// TIA Portal V17 export
// export: Created 2025-03-07T09:16:32.0834683Z, ExportSetting WithDefaults, DisplayName Totally Integrated Automation Portal, DisplayVersion V17 Update 8, DisplayName TIA Portal Openness, DisplayVersion V17 Update 8, DisplayName TIA Portal Version Control Interface, DisplayVersion V17, DisplayName SINAMICS Startdrive Advanced, DisplayVersion V17 SP2, DisplayName SINAMICS Startdrive G110M, G120, G120C, G120D, G120P, G115D, DisplayVersion V17 SP2, DisplayName SINAMICS Startdrive G130, G150, S120, S150, SINAMICS MV, S210, DisplayVersion V17 SP2, DisplayName STEP 7 Professional, DisplayVersion V17 Update 8, DisplayName SINUMERIK ONE STEP 7 Toolbox, DisplayVersion V17 Update 12, DisplayName SINUMERIK 840D sl STEP 7 Toolbox, DisplayVersion V17 Update 12, DisplayName STEP 7 Safety, DisplayVersion V17 Update 6, DisplayName WinCC Advanced, DisplayVersion V17 Update 8
DATA_BLOCK "LBP_ParamAlarmMsgs"   // DB5
TITLE = PLC-Error / Messages / PLC errores/avisos / PLC-Fehler / Meldungen
{ S7_Optimized_Access := 'FALSE'; DB_Accessible_From_OPC_UA := 'FALSE' }
AUTHOR : SINUMERIK
FAMILY : SINUMERIK_ONE
VERSION : 6.15
// Interface between user program and LBP_GenAlarmMsgs [FC10], contains the parameter assignment of the alarms for the bit arrays in the LBP_AlarmMsgs [DB2] as fault or status message. / Interfaz entre programa de usuario y LBP_GenAlarmMsgs [FC10], contiene la asignación de parámetros de las alarmas para los arrays de bits en LBP_AlarmMsgs [DB2] como avisos de fallo o de estado. / Schnittstelle zwischen Anwenderprogramm und LBP_GenAlarmMsgs [FC10], enthält die Parameterzuordnung der Alarme für die Bit-Arrays in der LBP_AlarmMsgs [DB2] als Störungs- oder Statusmeldungen.
// stored: AutoNumber false, DBAccessibleFromOPCUA false, DBAccessibleFromWebserver true, IsOnlyStoredInLoadMemory false, IsWriteProtectedInAS false
   VAR RETAIN
      Ch1_DB2_310 : Bool := TRUE;   // (Kanäle 1-10, je 18 Bit): DB2.DBB310; Fehlermeldungen / (Channels 1-10, 18 bits each): DB2.DBB310; error messages / (Canales 1-10, cada uno 18 bits): DB2.DBB310; avisos de error
      Ch1_DB2_311 : Bool := FALSE;   // Kanal 1, DB2.DBB311; Betriebsmeldungen / Channel 1, DB2.DBB311; operating messages / Canal 1, DB2.DBB311; avisos operativos
      Ch1_DB2_312 : Bool := TRUE;   // Kanal 1, DB2.DBB312; Fehlermeldungen / Channel 1, DB2.DBB312; error messages / Canal 1, DB2.DBB312; avisos de error
      Ch1_DB2_313 : Bool := TRUE;   // Fehlermeldungen / Error messages / Avisos de error
      Ch1_DB2_314 : Bool := FALSE;   // Betriebsmeldungen / Operating messages / Avisos operativos
      Ch1_DB2_315 : Bool := FALSE;   // Betriebsmeldungen / Operating messages / Avisos operativos
      Ch1_DB2_316 : Bool := TRUE;   // Fehlermeldungen / Error messages / Avisos de error
      Ch1_DB2_317 : Bool := TRUE;   // Fehlermeldungen / Error messages / Avisos de error
      Ch1_DB2_318 : Bool := FALSE;   // Betriebsmeldungen / Operating messages / Avisos operativos
      Ch1_DB2_319 : Bool := FALSE;   // Betriebsmeldungen / Operating messages / Avisos operativos
      Ch1_DB2_320 : Bool := TRUE;   // Fehlermeldungen / Error messages / Avisos de error
      Ch1_DB2_321 : Bool := FALSE;   // Betriebsmeldungen / Operating messages / Avisos operativos
      Ch1_DB2_322 : Bool := TRUE;   // Fehlermeldungen / Error messages / Avisos de error
      Ch1_DB2_323 : Bool := FALSE;   // Betriebsmeldungen / Operating messages / Avisos operativos
      Ch1_DB2_324 : Bool := TRUE;   // Fehlermeldungen / Error messages / Avisos de error
      Ch1_DB2_325 : Bool := FALSE;   // Betriebsmeldungen / Operating messages / Avisos operativos
      Ch1_DB2_326 : Bool := TRUE;   // Fehlermeldungen / Error messages / Avisos de error
      Ch1_DB2_327 : Bool := FALSE;   // Betriebsmeldungen / Operating messages / Avisos operativos
      Ch2_DB2_328 : Bool := TRUE;   // Kanal 2, DB2.DBB328; Fehlermeldungen / Channel 2, DB2.DBB328; error messages / Canal 2, DB2.DBB328; avisos de error
      Ch2_DB2_329 : Bool := FALSE;   // Kanal 2, DB2.DBB329; Betriebsmeldungen / Channel 2, DB2.DBB329; operating messages / Canal 2, DB2.DBB329; avisos operativos
      Ch2_DB2_330 : Bool := TRUE;   // Fehlermeldungen / Error messages / Avisos de error
      Ch2_DB2_331 : Bool := TRUE;   // Fehlermeldungen / Error messages / Avisos de error
      Ch2_DB2_332 : Bool := FALSE;   // Betriebsmeldungen / Operating messages / Avisos operativos
      Ch2_DB2_333 : Bool := FALSE;   // Betriebsmeldungen / Operating messages / Avisos operativos
      Ch2_DB2_334 : Bool := TRUE;   // Fehlermeldungen / Error messages / Avisos de error
      Ch2_DB2_335 : Bool := TRUE;   // Fehlermeldungen / Error messages / Avisos de error
      Ch2_DB2_336 : Bool := FALSE;   // Betriebsmeldungen / Operating messages / Avisos operativos
      Ch2_DB2_337 : Bool := FALSE;   // Betriebsmeldungen / Operating messages / Avisos operativos
      Ch2_DB2_338 : Bool := TRUE;   // Fehlermeldungen / Error messages / Avisos de error
      Ch2_DB2_339 : Bool := FALSE;   // Betriebsmeldungen / Operating messages / Avisos operativos
      Ch2_DB2_340 : Bool := TRUE;   // Fehlermeldungen / Error messages / Avisos de error
      Ch2_DB2_341 : Bool := FALSE;   // Betriebsmeldungen / Operating messages / Avisos operativos
      Ch2_DB2_342 : Bool := TRUE;   // Fehlermeldungen / Error messages / Avisos de error
      Ch2_DB2_343 : Bool := FALSE;   // Betriebsmeldungen / Operating messages / Avisos operativos
      Ch2_DB2_344 : Bool := TRUE;   // Fehlermeldungen / Error messages / Avisos de error
      Ch2_DB2_345 : Bool := FALSE;   // Betriebsmeldungen / Operating messages / Avisos operativos
      Ch3_DB2_346 : Bool := TRUE;   // Kanal 3, DB2.DBB346; Fehlermeldungen / Channel 3, DB2.DBB346; error messages / Canal 3, DB2.DBB346; avisos de error
      Ch3_DB2_347 : Bool := FALSE;   // Kanal 3, DB2.DBB347; Betriebsmeldungen / Channel 3, DB2.DBB347; operating messages / Canal 3, DB2.DBB347; avisos operativos
      Ch3_DB2_348 : Bool := TRUE;   // Fehlermeldungen / Error messages / Avisos de error
      Ch3_DB2_349 : Bool := TRUE;   // Fehlermeldungen / Error messages / Avisos de error
      Ch3_DB2_350 : Bool := FALSE;   // Betriebsmeldungen / Operating messages / Avisos operativos
      Ch3_DB2_351 : Bool := FALSE;   // Betriebsmeldungen / Operating messages / Avisos operativos
      Ch3_DB2_352 : Bool := TRUE;   // Fehlermeldungen / Error messages / Avisos de error
      Ch3_DB2_353 : Bool := TRUE;   // Fehlermeldungen / Error messages / Avisos de error
      Ch3_DB2_354 : Bool := FALSE;   // Betriebsmeldungen / Operating messages / Avisos operativos
      Ch3_DB2_355 : Bool := FALSE;   // Betriebsmeldungen / Operating messages / Avisos operativos
      Ch3_DB2_356 : Bool := TRUE;   // Fehlermeldungen / Error messages / Avisos de error
      Ch3_DB2_357 : Bool := FALSE;   // Betriebsmeldungen / Operating messages / Avisos operativos
      Ch3_DB2_358 : Bool := TRUE;   // Fehlermeldungen / Error messages / Avisos de error
      Ch3_DB2_359 : Bool := FALSE;   // Betriebsmeldungen / Operating messages / Avisos operativos
      Ch3_DB2_360 : Bool := TRUE;   // Fehlermeldungen / Error messages / Avisos de error
      Ch3_DB2_361 : Bool := FALSE;   // Betriebsmeldungen / Operating messages / Avisos operativos
      Ch3_DB2_362 : Bool := TRUE;   // Fehlermeldungen / Error messages / Avisos de error
      Ch3_DB2_363 : Bool := FALSE;   // Betriebsmeldungen / Operating messages / Avisos operativos
      Ch4_DB2_364 : Bool := TRUE;   // Kanal 4, DB2.DBB364; Fehlermeldungen / Channel 4, DB2.DBB364; error messages / Canal 4, DB2.DBB364; avisos de error
      Ch4_DB2_365 : Bool := FALSE;   // Kanal 4, DB2.DBB365; Betriebsmeldungen / Channel 4, DB2.DBB365; operating messages / Canal 4, DB2.DBB365; avisos operativos
      Ch4_DB2_366 : Bool := TRUE;   // Fehlermeldungen / Error messages / Avisos de error
      Ch4_DB2_367 : Bool := TRUE;   // Fehlermeldungen / Error messages / Avisos de error
      Ch4_DB2_368 : Bool := FALSE;   // Betriebsmeldungen / Operating messages / Avisos operativos
      Ch4_DB2_369 : Bool := FALSE;   // Betriebsmeldungen / Operating messages / Avisos operativos
      Ch4_DB2_370 : Bool := TRUE;   // Fehlermeldungen / Error messages / Avisos de error
      Ch4_DB2_371 : Bool := TRUE;   // Fehlermeldungen / Error messages / Avisos de error
      Ch4_DB2_372 : Bool := FALSE;   // Betriebsmeldungen / Operating messages / Avisos operativos
      Ch4_DB2_373 : Bool := FALSE;   // Betriebsmeldungen / Operating messages / Avisos operativos
      Ch4_DB2_374 : Bool := TRUE;   // Fehlermeldungen / Error messages / Avisos de error
      Ch4_DB2_375 : Bool := FALSE;   // Betriebsmeldungen / Operating messages / Avisos operativos
      Ch4_DB2_376 : Bool := TRUE;   // Fehlermeldungen / Error messages / Avisos de error
      Ch4_DB2_377 : Bool := FALSE;   // Betriebsmeldungen / Operating messages / Avisos operativos
      Ch4_DB2_378 : Bool := TRUE;   // Fehlermeldungen / Error messages / Avisos de error
      Ch4_DB2_379 : Bool := FALSE;   // Betriebsmeldungen / Operating messages / Avisos operativos
      Ch4_DB2_380 : Bool := TRUE;   // Fehlermeldungen / Error messages / Avisos de error
      Ch4_DB2_381 : Bool := FALSE;   // Betriebsmeldungen / Operating messages / Avisos operativos
      Ch5_DB2_382 : Bool := TRUE;   // Kanal 5, DB2.DBB382; Fehlermeldungen / Channel 5, DB2.DBB382; error messages / Canal 5, DB2.DBB382; avisos de error
      Ch5_DB2_383 : Bool := FALSE;   // Kanal 5, DB2.DBB383; Betriebsmeldungen / Channel 5, DB2.DBB383; operating messages / Canal 5, DB2.DBB383; avisos operativos
      Ch5_DB2_384 : Bool := TRUE;   // Fehlermeldungen / Error messages / Avisos de error
      Ch5_DB2_385 : Bool := TRUE;   // Fehlermeldungen / Error messages / Avisos de error
      Ch5_DB2_386 : Bool := FALSE;   // Betriebsmeldungen / Operating messages / Avisos operativos
      Ch5_DB2_387 : Bool := FALSE;   // Betriebsmeldungen / Operating messages / Avisos operativos
      Ch5_DB2_388 : Bool := TRUE;   // Fehlermeldungen / Error messages / Avisos de error
      Ch5_DB2_389 : Bool := TRUE;   // Fehlermeldungen / Error messages / Avisos de error
      Ch5_DB2_390 : Bool := FALSE;   // Betriebsmeldungen / Operating messages / Avisos operativos
      Ch5_DB2_391 : Bool := FALSE;   // Betriebsmeldungen / Operating messages / Avisos operativos
      Ch5_DB2_392 : Bool := TRUE;   // Fehlermeldungen / Error messages / Avisos de error
      Ch5_DB2_393 : Bool := FALSE;   // Betriebsmeldungen / Operating messages / Avisos operativos
      Ch5_DB2_394 : Bool := TRUE;   // Fehlermeldungen / Error messages / Avisos de error
      Ch5_DB2_395 : Bool := FALSE;   // Betriebsmeldungen / Operating messages / Avisos operativos
      Ch5_DB2_396 : Bool := TRUE;   // Fehlermeldungen / Error messages / Avisos de error
      Ch5_DB2_397 : Bool := FALSE;   // Betriebsmeldungen / Operating messages / Avisos operativos
      Ch5_DB2_398 : Bool := TRUE;   // Fehlermeldungen / Error messages / Avisos de error
      Ch5_DB2_399 : Bool := FALSE;   // Betriebsmeldungen / Operating messages / Avisos operativos
      Ch6_DB2_400 : Bool := TRUE;   // Kanal 6, DB2.DBB400; Fehlermeldungen / Channel 6, DB2.DBB400; error messages / Canal 6, DB2.DBB400; avisos de error
      Ch6_DB2_401 : Bool := FALSE;   // Kanal 6, DB2.DBB401; Betriebsmeldungen / Channel 6, DB2.DBB401; operating messages / Canal 6, DB2.DBB401; avisos operativos
      Ch6_DB2_402 : Bool := TRUE;   // Fehlermeldungen / Error messages / Avisos de error
      Ch6_DB2_403 : Bool := TRUE;   // Fehlermeldungen / Error messages / Avisos de error
      Ch6_DB2_404 : Bool := FALSE;   // Betriebsmeldungen / Operating messages / Avisos operativos
      Ch6_DB2_405 : Bool := FALSE;   // Betriebsmeldungen / Operating messages / Avisos operativos
      Ch6_DB2_406 : Bool := TRUE;   // Fehlermeldungen / Error messages / Avisos de error
      Ch6_DB2_407 : Bool := TRUE;   // Fehlermeldungen / Error messages / Avisos de error
      Ch6_DB2_408 : Bool := FALSE;   // Betriebsmeldungen / Operating messages / Avisos operativos
      Ch6_DB2_409 : Bool := FALSE;   // Betriebsmeldungen / Operating messages / Avisos operativos
      Ch6_DB2_410 : Bool := TRUE;   // Fehlermeldungen / Error messages / Avisos de error
      Ch6_DB2_411 : Bool := FALSE;   // Betriebsmeldungen / Operating messages / Avisos operativos
      Ch6_DB2_412 : Bool := TRUE;   // Fehlermeldungen / Error messages / Avisos de error
      Ch6_DB2_413 : Bool := FALSE;   // Betriebsmeldungen / Operating messages / Avisos operativos
      Ch6_DB2_414 : Bool := TRUE;   // Fehlermeldungen / Error messages / Avisos de error
      Ch6_DB2_415 : Bool := FALSE;   // Betriebsmeldungen / Operating messages / Avisos operativos
      Ch6_DB2_416 : Bool := TRUE;   // Fehlermeldungen / Error messages / Avisos de error
      Ch6_DB2_417 : Bool := FALSE;   // Betriebsmeldungen / Operating messages / Avisos operativos
      Ch7_DB2_418 : Bool := TRUE;   // Kanal 7, DB2.DBB418; Fehlermeldungen / Channel 7, DB2.DBB418; error messages / Canal 7, DB2.DBB418; avisos de error
      Ch7_DB2_419 : Bool := FALSE;   // Kanal 7, DB2.DBB419; Betriebsmeldungen / Channel 7, DB2.DBB419; operating messages / Canal 7, DB2.DBB419; avisos operativos
      Ch7_DB2_420 : Bool := TRUE;   // Fehlermeldungen / Error messages / Avisos de error
      Ch7_DB2_421 : Bool := TRUE;   // Fehlermeldungen / Error messages / Avisos de error
      Ch7_DB2_422 : Bool := FALSE;   // Betriebsmeldungen / Operating messages / Avisos operativos
      Ch7_DB2_423 : Bool := FALSE;   // Betriebsmeldungen / Operating messages / Avisos operativos
      Ch7_DB2_424 : Bool := TRUE;   // Fehlermeldungen / Error messages / Avisos de error
      Ch7_DB2_425 : Bool := TRUE;   // Fehlermeldungen / Error messages / Avisos de error
      Ch7_DB2_426 : Bool := FALSE;   // Betriebsmeldungen / Operating messages / Avisos operativos
      Ch7_DB2_427 : Bool := FALSE;   // Betriebsmeldungen / Operating messages / Avisos operativos
      Ch7_DB2_428 : Bool := TRUE;   // Fehlermeldungen / Error messages / Avisos de error
      Ch7_DB2_429 : Bool := FALSE;   // Betriebsmeldungen / Operating messages / Avisos operativos
      Ch7_DB2_430 : Bool := TRUE;   // Fehlermeldungen / Error messages / Avisos de error
      Ch7_DB2_431 : Bool := FALSE;   // Betriebsmeldungen / Operating messages / Avisos operativos
      Ch7_DB2_432 : Bool := TRUE;   // Fehlermeldungen / Error messages / Avisos de error
      Ch7_DB2_433 : Bool := FALSE;   // Betriebsmeldungen / Operating messages / Avisos operativos
      Ch7_DB2_434 : Bool := TRUE;   // Fehlermeldungen / Error messages / Avisos de error
      Ch7_DB2_435 : Bool := FALSE;   // Betriebsmeldungen / Operating messages / Avisos operativos
      Ch8_DB2_436 : Bool := TRUE;   // Kanal 8, DB2.DBB436; Fehlermeldungen / Channel 8, DB2.DBB436; error messages / Canal 8, DB2.DBB436; avisos de error
      Ch8_DB2_437 : Bool := FALSE;   // Kanal 8, DB2.DBB437; Betriebsmeldungen / Channel 8, DB2.DBB437; operating messages / Canal 8, DB2.DBB437; avisos operativos
      Ch8_DB2_438 : Bool := TRUE;   // Fehlermeldungen / Error messages / Avisos de error
      Ch8_DB2_439 : Bool := TRUE;   // Fehlermeldungen / Error messages / Avisos de error
      Ch8_DB2_440 : Bool := FALSE;   // Betriebsmeldungen / Operating messages / Avisos operativos
      Ch8_DB2_441 : Bool := FALSE;   // Betriebsmeldungen / Operating messages / Avisos operativos
      Ch8_DB2_442 : Bool := TRUE;   // Fehlermeldungen / Error messages / Avisos de error
      Ch8_DB2_443 : Bool := TRUE;   // Fehlermeldungen / Error messages / Avisos de error
      Ch8_DB2_444 : Bool := FALSE;   // Betriebsmeldungen / Operating messages / Avisos operativos
      Ch8_DB2_445 : Bool := FALSE;   // Betriebsmeldungen / Operating messages / Avisos operativos
      Ch8_DB2_446 : Bool := TRUE;   // Fehlermeldungen / Error messages / Avisos de error
      Ch8_DB2_447 : Bool := FALSE;   // Betriebsmeldungen / Operating messages / Avisos operativos
      Ch8_DB2_448 : Bool := TRUE;   // Fehlermeldungen / Error messages / Avisos de error
      Ch8_DB2_449 : Bool := FALSE;   // Betriebsmeldungen / Operating messages / Avisos operativos
      Ch8_DB2_450 : Bool := TRUE;   // Fehlermeldungen / Error messages / Avisos de error
      Ch8_DB2_451 : Bool := FALSE;   // Betriebsmeldungen / Operating messages / Avisos operativos
      Ch8_DB2_452 : Bool := TRUE;   // Fehlermeldungen / Error messages / Avisos de error
      Ch8_DB2_453 : Bool := FALSE;   // Betriebsmeldungen / Operating messages / Avisos operativos
      Ch9_DB2_454 : Bool := TRUE;   // Kanal 9, DB2.DBB454; Fehlermeldungen / Channel 9, DB2.DBB454; error messages / Canal 9, DB2.DBB454; avisos de error
      Ch9_DB2_455 : Bool := FALSE;   // Kanal 9, DB2.DBB455; Betriebsmeldungen / Channel 9, DB2.DBB455; operating messages / Canal 9, DB2.DBB455; avisos operativos
      Ch9_DB2_456 : Bool := TRUE;   // Fehlermeldungen / Error messages / Avisos de error
      Ch9_DB2_457 : Bool := TRUE;   // Fehlermeldungen / Error messages / Avisos de error
      Ch9_DB2_458 : Bool := FALSE;   // Betriebsmeldungen / Operating messages / Avisos operativos
      Ch9_DB2_459 : Bool := FALSE;   // Betriebsmeldungen / Operating messages / Avisos operativos
      Ch9_DB2_460 : Bool := TRUE;   // Fehlermeldungen / Error messages / Avisos de error
      Ch9_DB2_461 : Bool := TRUE;   // Fehlermeldungen / Error messages / Avisos de error
      Ch9_DB2_462 : Bool := FALSE;   // Betriebsmeldungen / Operating messages / Avisos operativos
      Ch9_DB2_463 : Bool := FALSE;   // Betriebsmeldungen / Operating messages / Avisos operativos
      Ch9_DB2_464 : Bool := TRUE;   // Fehlermeldungen / Error messages / Avisos de error
      Ch9_DB2_465 : Bool := FALSE;   // Betriebsmeldungen / Operating messages / Avisos operativos
      Ch9_DB2_466 : Bool := TRUE;   // Fehlermeldungen / Error messages / Avisos de error
      Ch9_DB2_467 : Bool := FALSE;   // Betriebsmeldungen / Operating messages / Avisos operativos
      Ch9_DB2_468 : Bool := TRUE;   // Fehlermeldungen / Error messages / Avisos de error
      Ch9_DB2_469 : Bool := FALSE;   // Betriebsmeldungen / Operating messages / Avisos operativos
      Ch9_DB2_470 : Bool := TRUE;   // Fehlermeldungen / Error messages / Avisos de error
      Ch9_DB2_471 : Bool := FALSE;   // Betriebsmeldungen / Operating messages / Avisos operativos
      Ch10_DB2_472 : Bool := TRUE;   // Kanal 10, DB2.DBB472; Fehlermeldungen / Channel 10, DB2.DBB472; error messages / Canal 10, DB2.DBB472; avisos de error
      Ch10_DB2_473 : Bool := FALSE;   // Kanal 10, DB2.DBB473; Betriebsmeldungen / Channel 10, DB2.DBB473; operating messages / Canal 10, DB2.DBB473; avisos operativos
      Ch10_DB2_474 : Bool := TRUE;   // Fehlermeldungen / Error messages / Avisos de error
      Ch10_DB2_475 : Bool := TRUE;   // Fehlermeldungen / Error messages / Avisos de error
      Ch10_DB2_476 : Bool := FALSE;   // Betriebsmeldungen / Operating messages / Avisos operativos
      Ch10_DB2_477 : Bool := FALSE;   // Betriebsmeldungen / Operating messages / Avisos operativos
      Ch10_DB2_478 : Bool := TRUE;   // Fehlermeldungen / Error messages / Avisos de error
      Ch10_DB2_479 : Bool := TRUE;   // Fehlermeldungen / Error messages / Avisos de error
      Ch10_DB2_480 : Bool := FALSE;   // Betriebsmeldungen / Operating messages / Avisos operativos
      Ch10_DB2_481 : Bool := FALSE;   // Betriebsmeldungen / Operating messages / Avisos operativos
      Ch10_DB2_482 : Bool := TRUE;   // Fehlermeldungen / Error messages / Avisos de error
      Ch10_DB2_483 : Bool := FALSE;   // Betriebsmeldungen / Operating messages / Avisos operativos
      Ch10_DB2_484 : Bool := TRUE;   // Fehlermeldungen / Error messages / Avisos de error
      Ch10_DB2_485 : Bool := FALSE;   // Betriebsmeldungen / Operating messages / Avisos operativos
      Ch10_DB2_486 : Bool := TRUE;   // Fehlermeldungen / Error messages / Avisos de error
      Ch10_DB2_487 : Bool := FALSE;   // Betriebsmeldungen / Operating messages / Avisos operativos
      Ch10_DB2_488 : Bool := TRUE;   // Fehlermeldungen / Error messages / Avisos de error
      Ch10_DB2_489 : Bool := FALSE;   // Betriebsmeldungen / Operating messages / Avisos operativos
      Ax1_DB2_490 : Bool := TRUE;   // (Achsen/Spindeln 1-31, je 2 Bit): DB2.DBB490; Fehlermeldungen / (Axes/Spindles 1-31, 2 bits each): DB2.DBB490; error messages / (Ejes/cabezales 1-31, cada uno 2 bits): DB2.DBB490; avisos de error
      Ax1_DB2_491 : Bool := FALSE;   // Achse/Spindel 1, DB2.DBB491; Betriebsmeldungen / Axis/Spindle 1, DB2.DBB491; operating messages / Eje/cabezal 1, DB2.DBB491; avisos operativos
      Ax2_DB2_492 : Bool := TRUE;   // Achse/Spindel 2, DB2.DBB492; Fehlermeldungen / Axis/Spindle 2, DB2.DBB492; error messages / Eje/cabezal 2, DB2.DBB492; avisos de error
      Ax2_DB2_493 : Bool := FALSE;   // Achse/Spindel 2, DB2.DBB493; Betriebsmeldungen / Axis/Spindle 2, DB2.DBB493; operating messages / Eje/cabezal 2, DB2.DBB493; avisos operativos
      Ax3_DB2_494 : Bool := TRUE;   // Fehlermeldungen / Error messages / Avisos de error
      Ax3_DB2_495 : Bool := FALSE;   // Betriebsmeldungen / Operating messages / Avisos operativos
      Ax4_DB2_496 : Bool := TRUE;   // Fehlermeldungen / Error messages / Avisos de error
      Ax4_DB2_497 : Bool := FALSE;   // Betriebsmeldungen / Operating messages / Avisos operativos
      Ax5_DB2_498 : Bool := TRUE;   // Fehlermeldungen / Error messages / Avisos de error
      Ax5_DB2_499 : Bool := FALSE;   // Betriebsmeldungen / Operating messages / Avisos operativos
      Ax6_DB2_500 : Bool := TRUE;   // Fehlermeldungen / Error messages / Avisos de error
      Ax6_DB2_501 : Bool := FALSE;   // Betriebsmeldungen / Operating messages / Avisos operativos
      Ax7_DB2_502 : Bool := TRUE;   // Fehlermeldungen / Error messages / Avisos de error
      Ax7_DB2_503 : Bool := FALSE;   // Betriebsmeldungen / Operating messages / Avisos operativos
      Ax8_DB2_504 : Bool := TRUE;   // Fehlermeldungen / Error messages / Avisos de error
      Ax8_DB2_505 : Bool := FALSE;   // Betriebsmeldungen / Operating messages / Avisos operativos
      Ax9_DB2_506 : Bool := TRUE;   // Fehlermeldungen / Error messages / Avisos de error
      Ax9_DB2_507 : Bool := FALSE;   // Betriebsmeldungen / Operating messages / Avisos operativos
      Ax10_DB2_508 : Bool := TRUE;   // Fehlermeldungen / Error messages / Avisos de error
      Ax10_DB2_509 : Bool := FALSE;   // Betriebsmeldungen / Operating messages / Avisos operativos
      Ax11_DB2_510 : Bool := TRUE;   // Fehlermeldungen / Error messages / Avisos de error
      Ax11_DB2_511 : Bool := FALSE;   // Betriebsmeldungen / Operating messages / Avisos operativos
      Ax12_DB2_512 : Bool := TRUE;   // Fehlermeldungen / Error messages / Avisos de error
      Ax12_DB2_513 : Bool := FALSE;   // Betriebsmeldungen / Operating messages / Avisos operativos
      Ax13_DB2_514 : Bool := TRUE;   // Fehlermeldungen / Error messages / Avisos de error
      Ax13_DB2_515 : Bool := FALSE;   // Betriebsmeldungen / Operating messages / Avisos operativos
      Ax14_DB2_516 : Bool := TRUE;   // Fehlermeldungen / Error messages / Avisos de error
      Ax14_DB2_517 : Bool := FALSE;   // Betriebsmeldungen / Operating messages / Avisos operativos
      Ax15_DB2_518 : Bool := TRUE;   // Fehlermeldungen / Error messages / Avisos de error
      Ax15_DB2_519 : Bool := FALSE;   // Betriebsmeldungen / Operating messages / Avisos operativos
      Ax16_DB2_520 : Bool := TRUE;   // Fehlermeldungen / Error messages / Avisos de error
      Ax16_DB2_521 : Bool := FALSE;   // Betriebsmeldungen / Operating messages / Avisos operativos
      Ax17_DB2_522 : Bool := TRUE;   // Fehlermeldungen / Error messages / Avisos de error
      Ax17_DB2_523 : Bool := FALSE;   // Betriebsmeldungen / Operating messages / Avisos operativos
      Ax18_DB2_524 : Bool := TRUE;   // Fehlermeldungen / Error messages / Avisos de error
      Ax18_DB2_525 : Bool := FALSE;   // Betriebsmeldungen / Operating messages / Avisos operativos
      Ax19_DB2_526 : Bool := TRUE;   // Fehlermeldungen / Error messages / Avisos de error
      Ax19_DB2_527 : Bool := FALSE;   // Betriebsmeldungen / Operating messages / Avisos operativos
      Ax20_DB2_528 : Bool := TRUE;   // Fehlermeldungen / Error messages / Avisos de error
      Ax20_DB2_529 : Bool := FALSE;   // Betriebsmeldungen / Operating messages / Avisos operativos
      Ax21_DB2_530 : Bool := TRUE;   // Fehlermeldungen / Error messages / Avisos de error
      Ax21_DB2_531 : Bool := FALSE;   // Betriebsmeldungen / Operating messages / Avisos operativos
      Ax22_DB2_532 : Bool := TRUE;   // Fehlermeldungen / Error messages / Avisos de error
      Ax22_DB2_533 : Bool := FALSE;   // Betriebsmeldungen / Operating messages / Avisos operativos
      Ax23_DB2_534 : Bool := TRUE;   // Fehlermeldungen / Error messages / Avisos de error
      Ax23_DB2_535 : Bool := FALSE;   // Betriebsmeldungen / Operating messages / Avisos operativos
      Ax24_DB2_536 : Bool := TRUE;   // Fehlermeldungen / Error messages / Avisos de error
      Ax24_DB2_537 : Bool := FALSE;   // Betriebsmeldungen / Operating messages / Avisos operativos
      Ax25_DB2_538 : Bool := TRUE;   // Fehlermeldungen / Error messages / Avisos de error
      Ax25_DB2_539 : Bool := FALSE;   // Betriebsmeldungen / Operating messages / Avisos operativos
      Ax26_DB2_540 : Bool := TRUE;   // Fehlermeldungen / Error messages / Avisos de error
      Ax26_DB2_541 : Bool := FALSE;   // Betriebsmeldungen / Operating messages / Avisos operativos
      Ax27_DB2_542 : Bool := TRUE;   // Fehlermeldungen / Error messages / Avisos de error
      Ax27_DB2_543 : Bool := FALSE;   // Betriebsmeldungen / Operating messages / Avisos operativos
      Ax28_DB2_544 : Bool := TRUE;   // Fehlermeldungen / Error messages / Avisos de error
      Ax28_DB2_545 : Bool := FALSE;   // Betriebsmeldungen / Operating messages / Avisos operativos
      Ax29_DB2_546 : Bool := TRUE;   // Fehlermeldungen / Error messages / Avisos de error
      Ax29_DB2_547 : Bool := FALSE;   // Betriebsmeldungen / Operating messages / Avisos operativos
      Ax30_DB2_548 : Bool := TRUE;   // Fehlermeldungen / Error messages / Avisos de error
      Ax30_DB2_549 : Bool := FALSE;   // Betriebsmeldungen / Operating messages / Avisos operativos
      Ax31_DB2_550 : Bool := TRUE;   // Fehlermeldungen / Error messages / Avisos de error
      Ax31_DB2_551 : Bool := FALSE;   // Betriebsmeldungen / Operating messages / Avisos operativos
      Bit30_2 : Bool := FALSE;   // Reserviert / Reserved / Reservado
      Bit30_3 : Bool := FALSE;   // Reserviert / Reserved / Reservado
      User0_DB2_554 : Bool := TRUE;   // (Anwender-Datenbereiche 0-31, je 8 Bit): DB2.DBB554; Fehlermeldungen / (User data areas 0-31, 8 bits each): DB2.DBB554; error messages / (Áreas de datos de usuario 0-31, cada una 8 bits): DB2.DBB554; avisos de error
      User0_DB2_555 : Bool := TRUE;   // UserDataArea 0, DB2.DBB555; Fehlermeldungen / UserDataArea 0, DB2.DBB555; error messages / UserDataArea 0, DB2.DBB555; avisos de error
      User0_DB2_556 : Bool := TRUE;   // Fehlermeldungen / Error messages / Avisos de error
      User0_DB2_557 : Bool := TRUE;   // Fehlermeldungen / Error messages / Avisos de error
      User0_DB2_558 : Bool := FALSE;   // Betriebsmeldungen / Operating messages / Avisos operativos
      User0_DB2_559 : Bool := FALSE;   // Betriebsmeldungen / Operating messages / Avisos operativos
      User0_DB2_560 : Bool := FALSE;   // Betriebsmeldungen / Operating messages / Avisos operativos
      User0_DB2_561 : Bool := FALSE;   // Betriebsmeldungen / Operating messages / Avisos operativos
      User1_DB2_562 : Bool := TRUE;   // UserDataArea 1, DB2.DBB562; Fehlermeldungen / UserDataArea 1, DB2.DBB562; error messages / UserDataArea 1, DB2.DBB562; avisos de error
      User1_DB2_563 : Bool := TRUE;   // Fehlermeldungen / Error messages / Avisos de error
      User1_DB2_564 : Bool := TRUE;   // Fehlermeldungen / Error messages / Avisos de error
      User1_DB2_565 : Bool := TRUE;   // Fehlermeldungen / Error messages / Avisos de error
      User1_DB2_566 : Bool := FALSE;   // Betriebsmeldungen / Operating messages / Avisos operativos
      User1_DB2_567 : Bool := FALSE;   // Betriebsmeldungen / Operating messages / Avisos operativos
      User1_DB2_568 : Bool := FALSE;   // Betriebsmeldungen / Operating messages / Avisos operativos
      User1_DB2_569 : Bool := FALSE;   // Betriebsmeldungen / Operating messages / Avisos operativos
      User2_DB2_570 : Bool := TRUE;   // UserDataArea 2, DB2.DBB570; Fehlermeldungen / UserDataArea 2, DB2.DBB570; error messages / UserDataArea 2, DB2.DBB570; avisos de error
      User2_DB2_571 : Bool := TRUE;   // Fehlermeldungen / Error messages / Avisos de error
      User2_DB2_572 : Bool := TRUE;   // Fehlermeldungen / Error messages / Avisos de error
      User2_DB2_573 : Bool := TRUE;   // Fehlermeldungen / Error messages / Avisos de error
      User2_DB2_574 : Bool := FALSE;   // Betriebsmeldungen / Operating messages / Avisos operativos
      User2_DB2_575 : Bool := FALSE;   // Betriebsmeldungen / Operating messages / Avisos operativos
      User2_DB2_576 : Bool := FALSE;   // Betriebsmeldungen / Operating messages / Avisos operativos
      User2_DB2_577 : Bool := FALSE;   // Betriebsmeldungen / Operating messages / Avisos operativos
      User3_DB2_578 : Bool := TRUE;   // UserDataArea 3, DB2.DBB578; Fehlermeldungen / UserDataArea 3, DB2.DBB578; error messages / UserDataArea 3, DB2.DBB578; avisos de error
      User3_DB2_579 : Bool := TRUE;   // Fehlermeldungen / Error messages / Avisos de error
      User3_DB2_580 : Bool := TRUE;   // Fehlermeldungen / Error messages / Avisos de error
      User3_DB2_581 : Bool := TRUE;   // Fehlermeldungen / Error messages / Avisos de error
      User3_DB2_582 : Bool := FALSE;   // Betriebsmeldungen / Operating messages / Avisos operativos
      User3_DB2_583 : Bool := FALSE;   // Betriebsmeldungen / Operating messages / Avisos operativos
      User3_DB2_584 : Bool := FALSE;   // Betriebsmeldungen / Operating messages / Avisos operativos
      User3_DB2_585 : Bool := FALSE;   // Betriebsmeldungen / Operating messages / Avisos operativos
      User4_DB2_586 : Bool := TRUE;   // UserDataArea 4, DB2.DBB586; Fehlermeldungen / UserDataArea 4, DB2.DBB586; error messages / UserDataArea 4, DB2.DBB586; avisos de error
      User4_DB2_587 : Bool := TRUE;   // Fehlermeldungen / Error messages / Avisos de error
      User4_DB2_588 : Bool := TRUE;   // Fehlermeldungen / Error messages / Avisos de error
      User4_DB2_589 : Bool := TRUE;   // Fehlermeldungen / Error messages / Avisos de error
      User4_DB2_590 : Bool := FALSE;   // Betriebsmeldungen / Operating messages / Avisos operativos
      User4_DB2_591 : Bool := FALSE;   // Betriebsmeldungen / Operating messages / Avisos operativos
      User4_DB2_592 : Bool := FALSE;   // Betriebsmeldungen / Operating messages / Avisos operativos
      User4_DB2_593 : Bool := FALSE;   // Betriebsmeldungen / Operating messages / Avisos operativos
      User5_DB2_594 : Bool := TRUE;   // UserDataArea 5, DB2.DBB594; Fehlermeldungen / UserDataArea 5, DB2.DBB594; error messages / UserDataArea 5, DB2.DBB594; avisos de error
      User5_DB2_595 : Bool := TRUE;   // Fehlermeldungen / Error messages / Avisos de error
      User5_DB2_596 : Bool := TRUE;   // Fehlermeldungen / Error messages / Avisos de error
      User5_DB2_597 : Bool := TRUE;   // Fehlermeldungen / Error messages / Avisos de error
      User5_DB2_598 : Bool := FALSE;   // Betriebsmeldungen / Operating messages / Avisos operativos
      User5_DB2_599 : Bool := FALSE;   // Betriebsmeldungen / Operating messages / Avisos operativos
      User5_DB2_600 : Bool := FALSE;   // Betriebsmeldungen / Operating messages / Avisos operativos
      User5_DB2_601 : Bool := FALSE;   // Betriebsmeldungen / Operating messages / Avisos operativos
      User6_DB2_602 : Bool := TRUE;   // UserDataArea 6, DB2.DBB602; Fehlermeldungen / UserDataArea 6, DB2.DBB602; error messages / UserDataArea 6, DB2.DBB602; avisos de error
      User6_DB2_603 : Bool := TRUE;   // Fehlermeldungen / Error messages / Avisos de error
      User6_DB2_604 : Bool := TRUE;   // Fehlermeldungen / Error messages / Avisos de error
      User6_DB2_605 : Bool := TRUE;   // Fehlermeldungen / Error messages / Avisos de error
      User6_DB2_606 : Bool := FALSE;   // Betriebsmeldungen / Operating messages / Avisos operativos
      User6_DB2_607 : Bool := FALSE;   // Betriebsmeldungen / Operating messages / Avisos operativos
      User6_DB2_608 : Bool := FALSE;   // Betriebsmeldungen / Operating messages / Avisos operativos
      User6_DB2_609 : Bool := FALSE;   // Betriebsmeldungen / Operating messages / Avisos operativos
      User7_DB2_610 : Bool := TRUE;   // UserDataArea 7, DB2.DBB610; Fehlermeldungen / UserDataArea 7, DB2.DBB610; error messages / UserDataArea 7, DB2.DBB610; avisos de error
      User7_DB2_611 : Bool := TRUE;   // Fehlermeldungen / Error messages / Avisos de error
      User7_DB2_612 : Bool := TRUE;   // Fehlermeldungen / Error messages / Avisos de error
      User7_DB2_613 : Bool := TRUE;   // Fehlermeldungen / Error messages / Avisos de error
      User7_DB2_614 : Bool := FALSE;   // Betriebsmeldungen / Operating messages / Avisos operativos
      User7_DB2_615 : Bool := FALSE;   // Betriebsmeldungen / Operating messages / Avisos operativos
      User7_DB2_616 : Bool := FALSE;   // Betriebsmeldungen / Operating messages / Avisos operativos
      User7_DB2_617 : Bool := FALSE;   // Betriebsmeldungen / Operating messages / Avisos operativos
      User8_DB2_618 : Bool := TRUE;   // UserDataArea 8, DB2.DBB618; Fehlermeldungen / UserDataArea 8, DB2.DBB618; error messages / UserDataArea 8, DB2.DBB618; avisos de error
      User8_DB2_619 : Bool := TRUE;   // Fehlermeldungen / Error messages / Avisos de error
      User8_DB2_620 : Bool := TRUE;   // Fehlermeldungen / Error messages / Avisos de error
      User8_DB2_621 : Bool := TRUE;   // Fehlermeldungen / Error messages / Avisos de error
      User8_DB2_622 : Bool := FALSE;   // Betriebsmeldungen / Operating messages / Avisos operativos
      User8_DB2_623 : Bool := FALSE;   // Betriebsmeldungen / Operating messages / Avisos operativos
      User8_DB2_624 : Bool := FALSE;   // Betriebsmeldungen / Operating messages / Avisos operativos
      User8_DB2_625 : Bool := FALSE;   // Betriebsmeldungen / Operating messages / Avisos operativos
      User9_DB2_626 : Bool := TRUE;   // UserDataArea 9, DB2.DBB626; Fehlermeldungen / UserDataArea 9, DB2.DBB626; error messages / UserDataArea 9, DB2.DBB626; avisos de error
      User9_DB2_627 : Bool := TRUE;   // Fehlermeldungen / Error messages / Avisos de error
      User9_DB2_628 : Bool := TRUE;   // Fehlermeldungen / Error messages / Avisos de error
      User9_DB2_629 : Bool := TRUE;   // Fehlermeldungen / Error messages / Avisos de error
      User9_DB2_630 : Bool := FALSE;   // Betriebsmeldungen / Operating messages / Avisos operativos
      User9_DB2_631 : Bool := FALSE;   // Betriebsmeldungen / Operating messages / Avisos operativos
      User9_DB2_632 : Bool := FALSE;   // Betriebsmeldungen / Operating messages / Avisos operativos
      User9_DB2_633 : Bool := FALSE;   // Betriebsmeldungen / Operating messages / Avisos operativos
      User10_DB2_634 : Bool := TRUE;   // UserDataArea 10, DB2.DBB634; Fehlermeldungen / UserDataArea 10, DB2.DBB634; error messages / UserDataArea 10, DB2.DBB634; avisos de error
      User10_DB2_635 : Bool := TRUE;   // Fehlermeldungen / Error messages / Avisos de error
      User10_DB2_636 : Bool := TRUE;   // Fehlermeldungen / Error messages / Avisos de error
      User10_DB2_637 : Bool := TRUE;   // Fehlermeldungen / Error messages / Avisos de error
      User10_DB2_638 : Bool := FALSE;   // Betriebsmeldungen / Operating messages / Avisos operativos
      User10_DB2_639 : Bool := FALSE;   // Betriebsmeldungen / Operating messages / Avisos operativos
      User10_DB2_640 : Bool := FALSE;   // Betriebsmeldungen / Operating messages / Avisos operativos
      User10_DB2_641 : Bool := FALSE;   // Betriebsmeldungen / Operating messages / Avisos operativos
      User11_DB2_642 : Bool := TRUE;   // UserDataArea 11, DB2.DBB642; Fehlermeldungen / UserDataArea 11, DB2.DBB642; error messages / UserDataArea 11, DB2.DBB642; avisos de error
      User11_DB2_643 : Bool := TRUE;   // Fehlermeldungen / Error messages / Avisos de error
      User11_DB2_644 : Bool := TRUE;   // Fehlermeldungen / Error messages / Avisos de error
      User11_DB2_645 : Bool := TRUE;   // Fehlermeldungen / Error messages / Avisos de error
      User11_DB2_646 : Bool := FALSE;   // Betriebsmeldungen / Operating messages / Avisos operativos
      User11_DB2_647 : Bool := FALSE;   // Betriebsmeldungen / Operating messages / Avisos operativos
      User11_DB2_648 : Bool := FALSE;   // Betriebsmeldungen / Operating messages / Avisos operativos
      User11_DB2_649 : Bool := FALSE;   // Betriebsmeldungen / Operating messages / Avisos operativos
      User12_DB2_650 : Bool := TRUE;   // UserDataArea 12, DB2.DBB650; Fehlermeldungen / UserDataArea 12, DB2.DBB650; error messages / UserDataArea 12, DB2.DBB650; avisos de error
      User12_DB2_651 : Bool := TRUE;   // Fehlermeldungen / Error messages / Avisos de error
      User12_DB2_652 : Bool := TRUE;   // Fehlermeldungen / Error messages / Avisos de error
      User12_DB2_653 : Bool := TRUE;   // Fehlermeldungen / Error messages / Avisos de error
      User12_DB2_654 : Bool := FALSE;   // Betriebsmeldungen / Operating messages / Avisos operativos
      User12_DB2_655 : Bool := FALSE;   // Betriebsmeldungen / Operating messages / Avisos operativos
      User12_DB2_656 : Bool := FALSE;   // Betriebsmeldungen / Operating messages / Avisos operativos
      User12_DB2_657 : Bool := FALSE;   // Betriebsmeldungen / Operating messages / Avisos operativos
      User13_DB2_658 : Bool := TRUE;   // UserDataArea 13, DB2.DBB658; Fehlermeldungen / UserDataArea 13, DB2.DBB658; error messages / UserDataArea 13, DB2.DBB658; avisos de error
      User13_DB2_659 : Bool := TRUE;   // Fehlermeldungen / Error messages / Avisos de error
      User13_DB2_660 : Bool := TRUE;   // Fehlermeldungen / Error messages / Avisos de error
      User13_DB2_661 : Bool := TRUE;   // Fehlermeldungen / Error messages / Avisos de error
      User13_DB2_662 : Bool := FALSE;   // Betriebsmeldungen / Operating messages / Avisos operativos
      User13_DB2_663 : Bool := FALSE;   // Betriebsmeldungen / Operating messages / Avisos operativos
      User13_DB2_664 : Bool := FALSE;   // Betriebsmeldungen / Operating messages / Avisos operativos
      User13_DB2_665 : Bool := FALSE;   // Betriebsmeldungen / Operating messages / Avisos operativos
      User14_DB2_666 : Bool := TRUE;   // UserDataArea 14, DB2.DBB666; Fehlermeldungen / UserDataArea 14, DB2.DBB666; error messages / UserDataArea 14, DB2.DBB666; avisos de error
      User14_DB2_667 : Bool := TRUE;   // Fehlermeldungen / Error messages / Avisos de error
      User14_DB2_668 : Bool := TRUE;   // Fehlermeldungen / Error messages / Avisos de error
      User14_DB2_669 : Bool := TRUE;   // Fehlermeldungen / Error messages / Avisos de error
      User14_DB2_670 : Bool := FALSE;   // Betriebsmeldungen / Operating messages / Avisos operativos
      User14_DB2_671 : Bool := FALSE;   // Betriebsmeldungen / Operating messages / Avisos operativos
      User14_DB2_672 : Bool := FALSE;   // Betriebsmeldungen / Operating messages / Avisos operativos
      User14_DB2_673 : Bool := FALSE;   // Betriebsmeldungen / Operating messages / Avisos operativos
      User15_DB2_674 : Bool := TRUE;   // UserDataArea 15, DB2.DBB674; Fehlermeldungen / UserDataArea 15, DB2.DBB674; error messages / UserDataArea 15, DB2.DBB674; avisos de error
      User15_DB2_675 : Bool := TRUE;   // Fehlermeldungen / Error messages / Avisos de error
      User15_DB2_676 : Bool := TRUE;   // Fehlermeldungen / Error messages / Avisos de error
      User15_DB2_677 : Bool := TRUE;   // Fehlermeldungen / Error messages / Avisos de error
      User15_DB2_678 : Bool := FALSE;   // Betriebsmeldungen / Operating messages / Avisos operativos
      User15_DB2_679 : Bool := FALSE;   // Betriebsmeldungen / Operating messages / Avisos operativos
      User15_DB2_680 : Bool := FALSE;   // Betriebsmeldungen / Operating messages / Avisos operativos
      User15_DB2_681 : Bool := FALSE;   // Betriebsmeldungen / Operating messages / Avisos operativos
      User16_DB2_682 : Bool := TRUE;   // UserDataArea 16, DB2.DBB682; Fehlermeldungen / UserDataArea 16, DB2.DBB682; error messages / UserDataArea 16, DB2.DBB682; avisos de error
      User16_DB2_683 : Bool := TRUE;   // Fehlermeldungen / Error messages / Avisos de error
      User16_DB2_684 : Bool := TRUE;   // Fehlermeldungen / Error messages / Avisos de error
      User16_DB2_685 : Bool := TRUE;   // Fehlermeldungen / Error messages / Avisos de error
      User16_DB2_686 : Bool := FALSE;   // Betriebsmeldungen / Operating messages / Avisos operativos
      User16_DB2_687 : Bool := FALSE;   // Betriebsmeldungen / Operating messages / Avisos operativos
      User16_DB2_688 : Bool := FALSE;   // Betriebsmeldungen / Operating messages / Avisos operativos
      User16_DB2_689 : Bool := FALSE;   // Betriebsmeldungen / Operating messages / Avisos operativos
      User17_DB2_690 : Bool := TRUE;   // UserDataArea 17, DB2.DBB690; Fehlermeldungen / UserDataArea 17, DB2.DBB690; error messages / UserDataArea 17, DB2.DBB690; avisos de error
      User17_DB2_691 : Bool := TRUE;   // Fehlermeldungen / Error messages / Avisos de error
      User17_DB2_692 : Bool := TRUE;   // Fehlermeldungen / Error messages / Avisos de error
      User17_DB2_693 : Bool := TRUE;   // Fehlermeldungen / Error messages / Avisos de error
      User17_DB2_694 : Bool := FALSE;   // Betriebsmeldungen / Operating messages / Avisos operativos
      User17_DB2_695 : Bool := FALSE;   // Betriebsmeldungen / Operating messages / Avisos operativos
      User17_DB2_696 : Bool := FALSE;   // Betriebsmeldungen / Operating messages / Avisos operativos
      User17_DB2_697 : Bool := FALSE;   // Betriebsmeldungen / Operating messages / Avisos operativos
      User18_DB2_698 : Bool := TRUE;   // UserDataArea 18, DB2.DBB698; Fehlermeldungen / UserDataArea 18, DB2.DBB698; error messages / UserDataArea 18, DB2.DBB698; avisos de error
      User18_DB2_699 : Bool := TRUE;   // Fehlermeldungen / Error messages / Avisos de error
      User18_DB2_700 : Bool := TRUE;   // Fehlermeldungen / Error messages / Avisos de error
      User18_DB2_701 : Bool := TRUE;   // Fehlermeldungen / Error messages / Avisos de error
      User18_DB2_702 : Bool := FALSE;   // Betriebsmeldungen / Operating messages / Avisos operativos
      User18_DB2_703 : Bool := FALSE;   // Betriebsmeldungen / Operating messages / Avisos operativos
      User18_DB2_704 : Bool := FALSE;   // Betriebsmeldungen / Operating messages / Avisos operativos
      User18_DB2_705 : Bool := FALSE;   // Betriebsmeldungen / Operating messages / Avisos operativos
      User19_DB2_706 : Bool := TRUE;   // UserDataArea 19, DB2.DBB706; Fehlermeldungen / UserDataArea 19, DB2.DBB706; error messages / UserDataArea 19, DB2.DBB706; avisos de error
      User19_DB2_707 : Bool := TRUE;   // Fehlermeldungen / Error messages / Avisos de error
      User19_DB2_708 : Bool := TRUE;   // Fehlermeldungen / Error messages / Avisos de error
      User19_DB2_709 : Bool := TRUE;   // Fehlermeldungen / Error messages / Avisos de error
      User19_DB2_710 : Bool := FALSE;   // Betriebsmeldungen / Operating messages / Avisos operativos
      User19_DB2_711 : Bool := FALSE;   // Betriebsmeldungen / Operating messages / Avisos operativos
      User19_DB2_712 : Bool := FALSE;   // Betriebsmeldungen / Operating messages / Avisos operativos
      User19_DB2_713 : Bool := FALSE;   // Betriebsmeldungen / Operating messages / Avisos operativos
      User20_DB2_714 : Bool := TRUE;   // UserDataArea 20, DB2.DBB714; Fehlermeldungen / UserDataArea 20, DB2.DBB714; error messages / UserDataArea 20, DB2.DBB714; avisos de error
      User20_DB2_715 : Bool := TRUE;   // Fehlermeldungen / Error messages / Avisos de error
      User20_DB2_716 : Bool := TRUE;   // Fehlermeldungen / Error messages / Avisos de error
      User20_DB2_717 : Bool := TRUE;   // Fehlermeldungen / Error messages / Avisos de error
      User20_DB2_718 : Bool := FALSE;   // Betriebsmeldungen / Operating messages / Avisos operativos
      User20_DB2_719 : Bool := FALSE;   // Betriebsmeldungen / Operating messages / Avisos operativos
      User20_DB2_720 : Bool := FALSE;   // Betriebsmeldungen / Operating messages / Avisos operativos
      User20_DB2_721 : Bool := FALSE;   // Betriebsmeldungen / Operating messages / Avisos operativos
      User21_DB2_722 : Bool := TRUE;   // UserDataArea 21, DB2.DBB722; Fehlermeldungen / UserDataArea 21, DB2.DBB722; error messages / UserDataArea 21, DB2.DBB722; avisos de error
      User21_DB2_723 : Bool := TRUE;   // Fehlermeldungen / Error messages / Avisos de error
      User21_DB2_724 : Bool := TRUE;   // Fehlermeldungen / Error messages / Avisos de error
      User21_DB2_725 : Bool := TRUE;   // Fehlermeldungen / Error messages / Avisos de error
      User21_DB2_726 : Bool := FALSE;   // Betriebsmeldungen / Operating messages / Avisos operativos
      User21_DB2_727 : Bool := FALSE;   // Betriebsmeldungen / Operating messages / Avisos operativos
      User21_DB2_728 : Bool := FALSE;   // Betriebsmeldungen / Operating messages / Avisos operativos
      User21_DB2_729 : Bool := FALSE;   // Betriebsmeldungen / Operating messages / Avisos operativos
      User22_DB2_730 : Bool := TRUE;   // UserDataArea 22, DB2.DBB730; Fehlermeldungen / UserDataArea 22, DB2.DBB730; error messages / UserDataArea 22, DB2.DBB730; avisos de error
      User22_DB2_731 : Bool := TRUE;   // Fehlermeldungen / Error messages / Avisos de error
      User22_DB2_732 : Bool := TRUE;   // Fehlermeldungen / Error messages / Avisos de error
      User22_DB2_733 : Bool := TRUE;   // Fehlermeldungen / Error messages / Avisos de error
      User22_DB2_734 : Bool := FALSE;   // Betriebsmeldungen / Operating messages / Avisos operativos
      User22_DB2_735 : Bool := FALSE;   // Betriebsmeldungen / Operating messages / Avisos operativos
      User22_DB2_736 : Bool := FALSE;   // Betriebsmeldungen / Operating messages / Avisos operativos
      User22_DB2_737 : Bool := FALSE;   // Betriebsmeldungen / Operating messages / Avisos operativos
      User23_DB2_738 : Bool := TRUE;   // UserDataArea 23, DB2.DBB738; Fehlermeldungen / UserDataArea 23, DB2.DBB738; error messages / UserDataArea 23, DB2.DBB738; avisos de error
      User23_DB2_739 : Bool := TRUE;   // Fehlermeldungen / Error messages / Avisos de error
      User23_DB2_740 : Bool := TRUE;   // Fehlermeldungen / Error messages / Avisos de error
      User23_DB2_741 : Bool := TRUE;   // Fehlermeldungen / Error messages / Avisos de error
      User23_DB2_742 : Bool := FALSE;   // Betriebsmeldungen / Operating messages / Avisos operativos
      User23_DB2_743 : Bool := FALSE;   // Betriebsmeldungen / Operating messages / Avisos operativos
      User23_DB2_744 : Bool := FALSE;   // Betriebsmeldungen / Operating messages / Avisos operativos
      User23_DB2_745 : Bool := FALSE;   // Betriebsmeldungen / Operating messages / Avisos operativos
      User24_DB2_746 : Bool := TRUE;   // UserDataArea 24, DB2.DBB746; Fehlermeldungen / UserDataArea 24, DB2.DBB746; error messages / UserDataArea 24, DB2.DBB746; avisos de error
      User24_DB2_747 : Bool := TRUE;   // Fehlermeldungen / Error messages / Avisos de error
      User24_DB2_748 : Bool := TRUE;   // Fehlermeldungen / Error messages / Avisos de error
      User24_DB2_749 : Bool := TRUE;   // Fehlermeldungen / Error messages / Avisos de error
      User24_DB2_750 : Bool := FALSE;   // Betriebsmeldungen / Operating messages / Avisos operativos
      User24_DB2_751 : Bool := FALSE;   // Betriebsmeldungen / Operating messages / Avisos operativos
      User24_DB2_752 : Bool := FALSE;   // Betriebsmeldungen / Operating messages / Avisos operativos
      User24_DB2_753 : Bool := FALSE;   // Betriebsmeldungen / Operating messages / Avisos operativos
      User25_DB2_754 : Bool := TRUE;   // UserDataArea 25, DB2.DBB754; Fehlermeldungen / UserDataArea 25, DB2.DBB754; error messages / UserDataArea 25, DB2.DBB754; avisos de error
      User25_DB2_755 : Bool := TRUE;   // Fehlermeldungen / Error messages / Avisos de error
      User25_DB2_756 : Bool := TRUE;   // Fehlermeldungen / Error messages / Avisos de error
      User25_DB2_757 : Bool := TRUE;   // Fehlermeldungen / Error messages / Avisos de error
      User25_DB2_758 : Bool := FALSE;   // Betriebsmeldungen / Operating messages / Avisos operativos
      User25_DB2_759 : Bool := FALSE;   // Betriebsmeldungen / Operating messages / Avisos operativos
      User25_DB2_760 : Bool := FALSE;   // Betriebsmeldungen / Operating messages / Avisos operativos
      User25_DB2_761 : Bool := FALSE;   // Betriebsmeldungen / Operating messages / Avisos operativos
      User26_DB2_762 : Bool := TRUE;   // UserDataArea 26, DB2.DBB762; Fehlermeldungen / UserDataArea 26, DB2.DBB762; error messages / UserDataArea 26, DB2.DBB762; avisos de error
      User26_DB2_763 : Bool := TRUE;   // Fehlermeldungen / Error messages / Avisos de error
      User26_DB2_764 : Bool := TRUE;   // Fehlermeldungen / Error messages / Avisos de error
      User26_DB2_765 : Bool := TRUE;   // Fehlermeldungen / Error messages / Avisos de error
      User26_DB2_766 : Bool := FALSE;   // Betriebsmeldungen / Operating messages / Avisos operativos
      User26_DB2_767 : Bool := FALSE;   // Betriebsmeldungen / Operating messages / Avisos operativos
      User26_DB2_768 : Bool := FALSE;   // Betriebsmeldungen / Operating messages / Avisos operativos
      User26_DB2_769 : Bool := FALSE;   // Betriebsmeldungen / Operating messages / Avisos operativos
      User27_DB2_770 : Bool := TRUE;   // UserDataArea 27, DB2.DBB770; Fehlermeldungen / UserDataArea 27, DB2.DBB770; error messages / UserDataArea 27, DB2.DBB770; avisos de error
      User27_DB2_771 : Bool := TRUE;   // Fehlermeldungen / Error messages / Avisos de error
      User27_DB2_772 : Bool := TRUE;   // Fehlermeldungen / Error messages / Avisos de error
      User27_DB2_773 : Bool := TRUE;   // Fehlermeldungen / Error messages / Avisos de error
      User27_DB2_774 : Bool := FALSE;   // Betriebsmeldungen / Operating messages / Avisos operativos
      User27_DB2_775 : Bool := FALSE;   // Betriebsmeldungen / Operating messages / Avisos operativos
      User27_DB2_776 : Bool := FALSE;   // Betriebsmeldungen / Operating messages / Avisos operativos
      User27_DB2_777 : Bool := FALSE;   // Betriebsmeldungen / Operating messages / Avisos operativos
      User28_DB2_778 : Bool := TRUE;   // UserDataArea 28, DB2.DBB778; Fehlermeldungen / UserDataArea 28, DB2.DBB778; error messages / UserDataArea 28, DB2.DBB778; avisos de error
      User28_DB2_779 : Bool := TRUE;   // Fehlermeldungen / Error messages / Avisos de error
      User28_DB2_780 : Bool := TRUE;   // Fehlermeldungen / Error messages / Avisos de error
      User28_DB2_781 : Bool := TRUE;   // Fehlermeldungen / Error messages / Avisos de error
      User28_DB2_782 : Bool := FALSE;   // Betriebsmeldungen / Operating messages / Avisos operativos
      User28_DB2_783 : Bool := FALSE;   // Betriebsmeldungen / Operating messages / Avisos operativos
      User28_DB2_784 : Bool := FALSE;   // Betriebsmeldungen / Operating messages / Avisos operativos
      User28_DB2_785 : Bool := FALSE;   // Betriebsmeldungen / Operating messages / Avisos operativos
      User29_DB2_786 : Bool := TRUE;   // UserDataArea 29, DB2.DBB786; Fehlermeldungen / UserDataArea 29, DB2.DBB786; error messages / UserDataArea 29, DB2.DBB786; avisos de error
      User29_DB2_787 : Bool := TRUE;   // Fehlermeldungen / Error messages / Avisos de error
      User29_DB2_788 : Bool := TRUE;   // Fehlermeldungen / Error messages / Avisos de error
      User29_DB2_789 : Bool := TRUE;   // Fehlermeldungen / Error messages / Avisos de error
      User29_DB2_790 : Bool := FALSE;   // Betriebsmeldungen / Operating messages / Avisos operativos
      User29_DB2_791 : Bool := FALSE;   // Betriebsmeldungen / Operating messages / Avisos operativos
      User29_DB2_792 : Bool := FALSE;   // Betriebsmeldungen / Operating messages / Avisos operativos
      User29_DB2_793 : Bool := FALSE;   // Betriebsmeldungen / Operating messages / Avisos operativos
      User30_DB2_794 : Bool := TRUE;   // UserDataArea 30, DB2.DBB794; Fehlermeldungen / UserDataArea 30, DB2.DBB794; error messages / UserDataArea 30, DB2.DBB794; avisos de error
      User30_DB2_795 : Bool := TRUE;   // Fehlermeldungen / Error messages / Avisos de error
      User30_DB2_796 : Bool := TRUE;   // Fehlermeldungen / Error messages / Avisos de error
      User30_DB2_797 : Bool := TRUE;   // Fehlermeldungen / Error messages / Avisos de error
      User30_DB2_798 : Bool := FALSE;   // Betriebsmeldungen / Operating messages / Avisos operativos
      User30_DB2_799 : Bool := FALSE;   // Betriebsmeldungen / Operating messages / Avisos operativos
      User30_DB2_800 : Bool := FALSE;   // Betriebsmeldungen / Operating messages / Avisos operativos
      User30_DB2_801 : Bool := FALSE;   // Betriebsmeldungen / Operating messages / Avisos operativos
      User31_DB2_802 : Bool := TRUE;   // UserDataArea 31, DB2.DBB802; Fehlermeldungen / UserDataArea 31, DB2.DBB802; error messages / UserDataArea 31, DB2.DBB802; avisos de error
      User31_DB2_803 : Bool := TRUE;   // Fehlermeldungen / Error messages / Avisos de error
      User31_DB2_804 : Bool := TRUE;   // Fehlermeldungen / Error messages / Avisos de error
      User31_DB2_805 : Bool := TRUE;   // Fehlermeldungen / Error messages / Avisos de error
      User31_DB2_806 : Bool := FALSE;   // Betriebsmeldungen / Operating messages / Avisos operativos
      User31_DB2_807 : Bool := FALSE;   // Betriebsmeldungen / Operating messages / Avisos operativos
      User31_DB2_808 : Bool := FALSE;   // Betriebsmeldungen / Operating messages / Avisos operativos
      User31_DB2_809 : Bool := FALSE;   // Betriebsmeldungen / Operating messages / Avisos operativos
      Bit62_4 : Bool;   // Reserviert / Reserved / Reservado
      Bit62_5 : Bool;   // Reserviert / Reserved / Reservado
      Bit62_6 : Bool;   // Reserviert / Reserved / Reservado
      Bit62_7 : Bool;   // Reserviert / Reserved / Reservado
      Byte63 : Byte;   // Reserviert / Reserved / Reservado
      Word64 : Word;   // Reserviert / Reserved / Reservado
      Word66 : Word;   // Reserviert / Reserved / Reservado
      Word68 : Word;   // Reserviert / Reserved / Reservado
      Word70 : Word;   // Reserviert / Reserved / Reservado
      ByteArray72 : Array[0..63] of Byte;   // Reserviert / Reserved / Reservado
      User32_DB2_810 : Bool := TRUE;   // (Anwender-Datenbereiche 32-63, je 8 Bit): DB2.DBB810; Fehlermeldungen / (User data areas 32-63, 8 bits each): DB2.DBB810; error messages / (Áreas de datos de usuario 32-63, cada una 8 bits): DB2.DBB810; avisos de error
      User32_DB2_811 : Bool := TRUE;   // Fehlermeldungen / Error messages / Avisos de error
      User32_DB2_812 : Bool := TRUE;   // Fehlermeldungen / Error messages / Avisos de error
      User32_DB2_813 : Bool := TRUE;   // Fehlermeldungen / Error messages / Avisos de error
      User32_DB2_814 : Bool := FALSE;   // Betriebsmeldungen / Operating messages / Avisos operativos
      User32_DB2_815 : Bool := FALSE;   // Betriebsmeldungen / Operating messages / Avisos operativos
      User32_DB2_816 : Bool := FALSE;   // Betriebsmeldungen / Operating messages / Avisos operativos
      User32_DB2_817 : Bool := FALSE;   // Betriebsmeldungen / Operating messages / Avisos operativos
      User33_DB2_818 : Bool := TRUE;   // UserDataArea 33, DB2.DBB818; Fehlermeldungen / UserDataArea 33, DB2.DBB818; error messages / UserDataArea 33, DB2.DBB818; avisos de error
      User33_DB2_819 : Bool := TRUE;   // Fehlermeldungen / Error messages / Avisos de error
      User33_DB2_820 : Bool := TRUE;   // Fehlermeldungen / Error messages / Avisos de error
      User33_DB2_821 : Bool := TRUE;   // Fehlermeldungen / Error messages / Avisos de error
      User33_DB2_822 : Bool := FALSE;   // Betriebsmeldungen / Operating messages / Avisos operativos
      User33_DB2_823 : Bool := FALSE;   // Betriebsmeldungen / Operating messages / Avisos operativos
      User33_DB2_824 : Bool := FALSE;   // Betriebsmeldungen / Operating messages / Avisos operativos
      User33_DB2_825 : Bool := FALSE;   // Betriebsmeldungen / Operating messages / Avisos operativos
      User34_DB2_826 : Bool := TRUE;   // UserDataArea 34, DB2.DBB826; Fehlermeldungen / UserDataArea 34, DB2.DBB826; error messages / UserDataArea 34, DB2.DBB826; avisos de error
      User34_DB2_827 : Bool := TRUE;   // Fehlermeldungen / Error messages / Avisos de error
      User34_DB2_828 : Bool := TRUE;   // Fehlermeldungen / Error messages / Avisos de error
      User34_DB2_829 : Bool := TRUE;   // Fehlermeldungen / Error messages / Avisos de error
      User34_DB2_830 : Bool := FALSE;   // Betriebsmeldungen / Operating messages / Avisos operativos
      User34_DB2_831 : Bool := FALSE;   // Betriebsmeldungen / Operating messages / Avisos operativos
      User34_DB2_832 : Bool := FALSE;   // Betriebsmeldungen / Operating messages / Avisos operativos
      User34_DB2_833 : Bool := FALSE;   // Betriebsmeldungen / Operating messages / Avisos operativos
      User35_DB2_834 : Bool := TRUE;   // UserDataArea 35, DB2.DBB834; Fehlermeldungen / UserDataArea 35, DB2.DBB834; error messages / UserDataArea 35, DB2.DBB834; avisos de error
      User35_DB2_835 : Bool := TRUE;   // Fehlermeldungen / Error messages / Avisos de error
      User35_DB2_836 : Bool := TRUE;   // Fehlermeldungen / Error messages / Avisos de error
      User35_DB2_837 : Bool := TRUE;   // Fehlermeldungen / Error messages / Avisos de error
      User35_DB2_838 : Bool := FALSE;   // Betriebsmeldungen / Operating messages / Avisos operativos
      User35_DB2_839 : Bool := FALSE;   // Betriebsmeldungen / Operating messages / Avisos operativos
      User35_DB2_840 : Bool := FALSE;   // Betriebsmeldungen / Operating messages / Avisos operativos
      User35_DB2_841 : Bool := FALSE;   // Betriebsmeldungen / Operating messages / Avisos operativos
      User36_DB2_842 : Bool := TRUE;   // UserDataArea 36, DB2.DBB842; Fehlermeldungen / UserDataArea 36, DB2.DBB842; error messages / UserDataArea 36, DB2.DBB842; avisos de error
      User36_DB2_843 : Bool := TRUE;   // Fehlermeldungen / Error messages / Avisos de error
      User36_DB2_844 : Bool := TRUE;   // Fehlermeldungen / Error messages / Avisos de error
      User36_DB2_845 : Bool := TRUE;   // Fehlermeldungen / Error messages / Avisos de error
      User36_DB2_846 : Bool := FALSE;   // Betriebsmeldungen / Operating messages / Avisos operativos
      User36_DB2_847 : Bool := FALSE;   // Betriebsmeldungen / Operating messages / Avisos operativos
      User36_DB2_848 : Bool := FALSE;   // Betriebsmeldungen / Operating messages / Avisos operativos
      User36_DB2_849 : Bool := FALSE;   // Betriebsmeldungen / Operating messages / Avisos operativos
      User37_DB2_850 : Bool := TRUE;   // UserDataArea 37, DB2.DBB850; Fehlermeldungen / UserDataArea 37, DB2.DBB850; error messages / UserDataArea 37, DB2.DBB850; avisos de error
      User37_DB2_851 : Bool := TRUE;   // Fehlermeldungen / Error messages / Avisos de error
      User37_DB2_852 : Bool := TRUE;   // Fehlermeldungen / Error messages / Avisos de error
      User37_DB2_853 : Bool := TRUE;   // Fehlermeldungen / Error messages / Avisos de error
      User37_DB2_854 : Bool := FALSE;   // Betriebsmeldungen / Operating messages / Avisos operativos
      User37_DB2_855 : Bool := FALSE;   // Betriebsmeldungen / Operating messages / Avisos operativos
      User37_DB2_856 : Bool := FALSE;   // Betriebsmeldungen / Operating messages / Avisos operativos
      User37_DB2_857 : Bool := FALSE;   // Betriebsmeldungen / Operating messages / Avisos operativos
      User38_DB2_858 : Bool := TRUE;   // UserDataArea 38, DB2.DBB858; Fehlermeldungen / UserDataArea 38, DB2.DBB858; error messages / UserDataArea 38, DB2.DBB858; avisos de error
      User38_DB2_859 : Bool := TRUE;   // Fehlermeldungen / Error messages / Avisos de error
      User38_DB2_860 : Bool := TRUE;   // Fehlermeldungen / Error messages / Avisos de error
      User38_DB2_861 : Bool := TRUE;   // Fehlermeldungen / Error messages / Avisos de error
      User38_DB2_862 : Bool := FALSE;   // Betriebsmeldungen / Operating messages / Avisos operativos
      User38_DB2_863 : Bool := FALSE;   // Betriebsmeldungen / Operating messages / Avisos operativos
      User38_DB2_864 : Bool := FALSE;   // Betriebsmeldungen / Operating messages / Avisos operativos
      User38_DB2_865 : Bool := FALSE;   // Betriebsmeldungen / Operating messages / Avisos operativos
      User39_DB2_866 : Bool := TRUE;   // UserDataArea 39, DB2.DBB866; Fehlermeldungen / UserDataArea 39, DB2.DBB866; error messages / UserDataArea 39, DB2.DBB866; avisos de error
      User39_DB2_867 : Bool := TRUE;   // Fehlermeldungen / Error messages / Avisos de error
      User39_DB2_868 : Bool := TRUE;   // Fehlermeldungen / Error messages / Avisos de error
      User39_DB2_869 : Bool := TRUE;   // Fehlermeldungen / Error messages / Avisos de error
      User39_DB2_870 : Bool := FALSE;   // Betriebsmeldungen / Operating messages / Avisos operativos
      User39_DB2_871 : Bool := FALSE;   // Betriebsmeldungen / Operating messages / Avisos operativos
      User39_DB2_872 : Bool := FALSE;   // Betriebsmeldungen / Operating messages / Avisos operativos
      User39_DB2_873 : Bool := FALSE;   // Betriebsmeldungen / Operating messages / Avisos operativos
      User40_DB2_874 : Bool := TRUE;   // UserDataArea 40, DB2.DBB874; Fehlermeldungen / UserDataArea 40, DB2.DBB874; error messages / UserDataArea 40, DB2.DBB874; avisos de error
      User40_DB2_875 : Bool := TRUE;   // Fehlermeldungen / Error messages / Avisos de error
      User40_DB2_876 : Bool := TRUE;   // Fehlermeldungen / Error messages / Avisos de error
      User40_DB2_877 : Bool := TRUE;   // Fehlermeldungen / Error messages / Avisos de error
      User40_DB2_878 : Bool := FALSE;   // Betriebsmeldungen / Operating messages / Avisos operativos
      User40_DB2_879 : Bool := FALSE;   // Betriebsmeldungen / Operating messages / Avisos operativos
      User40_DB2_880 : Bool := FALSE;   // Betriebsmeldungen / Operating messages / Avisos operativos
      User40_DB2_881 : Bool := FALSE;   // Betriebsmeldungen / Operating messages / Avisos operativos
      User41_DB2_882 : Bool := TRUE;   // UserDataArea 41, DB2.DBB882; Fehlermeldungen / UserDataArea 41, DB2.DBB882; error messages / UserDataArea 41, DB2.DBB882; avisos de error
      User41_DB2_883 : Bool := TRUE;   // Fehlermeldungen / Error messages / Avisos de error
      User41_DB2_884 : Bool := TRUE;   // Fehlermeldungen / Error messages / Avisos de error
      User41_DB2_885 : Bool := TRUE;   // Fehlermeldungen / Error messages / Avisos de error
      User41_DB2_886 : Bool := FALSE;   // Betriebsmeldungen / Operating messages / Avisos operativos
      User41_DB2_887 : Bool := FALSE;   // Betriebsmeldungen / Operating messages / Avisos operativos
      User41_DB2_888 : Bool := FALSE;   // Betriebsmeldungen / Operating messages / Avisos operativos
      User41_DB2_889 : Bool := FALSE;   // Betriebsmeldungen / Operating messages / Avisos operativos
      User42_DB2_890 : Bool := TRUE;   // UserDataArea 42, DB2.DBB890; Fehlermeldungen / UserDataArea 42, DB2.DBB890; error messages / UserDataArea 42, DB2.DBB890; avisos de error
      User42_DB2_891 : Bool := TRUE;   // Fehlermeldungen / Error messages / Avisos de error
      User42_DB2_892 : Bool := TRUE;   // Fehlermeldungen / Error messages / Avisos de error
      User42_DB2_893 : Bool := TRUE;   // Fehlermeldungen / Error messages / Avisos de error
      User42_DB2_894 : Bool := FALSE;   // Betriebsmeldungen / Operating messages / Avisos operativos
      User42_DB2_895 : Bool := FALSE;   // Betriebsmeldungen / Operating messages / Avisos operativos
      User42_DB2_896 : Bool := FALSE;   // Betriebsmeldungen / Operating messages / Avisos operativos
      User42_DB2_897 : Bool := FALSE;   // Betriebsmeldungen / Operating messages / Avisos operativos
      User43_DB2_898 : Bool := TRUE;   // UserDataArea 43, DB2.DBB898; Fehlermeldungen / UserDataArea 43, DB2.DBB898; error messages / UserDataArea 43, DB2.DBB898; avisos de error
      User43_DB2_899 : Bool := TRUE;   // Fehlermeldungen / Error messages / Avisos de error
      User43_DB2_900 : Bool := TRUE;   // Fehlermeldungen / Error messages / Avisos de error
      User43_DB2_901 : Bool := TRUE;   // Fehlermeldungen / Error messages / Avisos de error
      User43_DB2_902 : Bool := FALSE;   // Betriebsmeldungen / Operating messages / Avisos operativos
      User43_DB2_903 : Bool := FALSE;   // Betriebsmeldungen / Operating messages / Avisos operativos
      User43_DB2_904 : Bool := FALSE;   // Betriebsmeldungen / Operating messages / Avisos operativos
      User43_DB2_905 : Bool := FALSE;   // Betriebsmeldungen / Operating messages / Avisos operativos
      User44_DB2_906 : Bool := TRUE;   // UserDataArea 44, DB2.DBB906; Fehlermeldungen / UserDataArea 44, DB2.DBB906; error messages / UserDataArea 44, DB2.DBB906; avisos de error
      User44_DB2_907 : Bool := TRUE;   // Fehlermeldungen / Error messages / Avisos de error
      User44_DB2_908 : Bool := TRUE;   // Fehlermeldungen / Error messages / Avisos de error
      User44_DB2_909 : Bool := TRUE;   // Fehlermeldungen / Error messages / Avisos de error
      User44_DB2_910 : Bool := FALSE;   // Betriebsmeldungen / Operating messages / Avisos operativos
      User44_DB2_911 : Bool := FALSE;   // Betriebsmeldungen / Operating messages / Avisos operativos
      User44_DB2_912 : Bool := FALSE;   // Betriebsmeldungen / Operating messages / Avisos operativos
      User44_DB2_913 : Bool := FALSE;   // Betriebsmeldungen / Operating messages / Avisos operativos
      User45_DB2_914 : Bool := TRUE;   // UserDataArea 45, DB2.DBB914; Fehlermeldungen / UserDataArea 45, DB2.DBB914; error messages / UserDataArea 45, DB2.DBB914; avisos de error
      User45_DB2_915 : Bool := TRUE;   // Fehlermeldungen / Error messages / Avisos de error
      User45_DB2_916 : Bool := TRUE;   // Fehlermeldungen / Error messages / Avisos de error
      User45_DB2_917 : Bool := TRUE;   // Fehlermeldungen / Error messages / Avisos de error
      User45_DB2_918 : Bool := FALSE;   // Betriebsmeldungen / Operating messages / Avisos operativos
      User45_DB2_919 : Bool := FALSE;   // Betriebsmeldungen / Operating messages / Avisos operativos
      User45_DB2_920 : Bool := FALSE;   // Betriebsmeldungen / Operating messages / Avisos operativos
      User45_DB2_921 : Bool := FALSE;   // Betriebsmeldungen / Operating messages / Avisos operativos
      User46_DB2_922 : Bool := TRUE;   // UserDataArea 46, DB2.DBB922; Fehlermeldungen / UserDataArea 46, DB2.DBB922; error messages / UserDataArea 46, DB2.DBB922; avisos de error
      User46_DB2_923 : Bool := TRUE;   // Fehlermeldungen / Error messages / Avisos de error
      User46_DB2_924 : Bool := TRUE;   // Fehlermeldungen / Error messages / Avisos de error
      User46_DB2_925 : Bool := TRUE;   // Fehlermeldungen / Error messages / Avisos de error
      User46_DB2_926 : Bool := FALSE;   // Betriebsmeldungen / Operating messages / Avisos operativos
      User46_DB2_927 : Bool := FALSE;   // Betriebsmeldungen / Operating messages / Avisos operativos
      User46_DB2_928 : Bool := FALSE;   // Betriebsmeldungen / Operating messages / Avisos operativos
      User46_DB2_929 : Bool := FALSE;   // Betriebsmeldungen / Operating messages / Avisos operativos
      User47_DB2_930 : Bool := TRUE;   // UserDataArea 47, DB2.DBB930; Fehlermeldungen / UserDataArea 47, DB2.DBB930; error messages / UserDataArea 47, DB2.DBB930; avisos de error
      User47_DB2_931 : Bool := TRUE;   // Fehlermeldungen / Error messages / Avisos de error
      User47_DB2_932 : Bool := TRUE;   // Fehlermeldungen / Error messages / Avisos de error
      User47_DB2_933 : Bool := TRUE;   // Fehlermeldungen / Error messages / Avisos de error
      User47_DB2_934 : Bool := FALSE;   // Betriebsmeldungen / Operating messages / Avisos operativos
      User47_DB2_935 : Bool := FALSE;   // Betriebsmeldungen / Operating messages / Avisos operativos
      User47_DB2_936 : Bool := FALSE;   // Betriebsmeldungen / Operating messages / Avisos operativos
      User47_DB2_937 : Bool := FALSE;   // Betriebsmeldungen / Operating messages / Avisos operativos
      User48_DB2_938 : Bool := TRUE;   // UserDataArea 48, DB2.DBB938; Fehlermeldungen / UserDataArea 48, DB2.DBB938; error messages / UserDataArea 48, DB2.DBB938; avisos de error
      User48_DB2_939 : Bool := TRUE;   // Fehlermeldungen / Error messages / Avisos de error
      User48_DB2_940 : Bool := TRUE;   // Fehlermeldungen / Error messages / Avisos de error
      User48_DB2_941 : Bool := TRUE;   // Fehlermeldungen / Error messages / Avisos de error
      User48_DB2_942 : Bool := FALSE;   // Betriebsmeldungen / Operating messages / Avisos operativos
      User48_DB2_943 : Bool := FALSE;   // Betriebsmeldungen / Operating messages / Avisos operativos
      User48_DB2_944 : Bool := FALSE;   // Betriebsmeldungen / Operating messages / Avisos operativos
      User48_DB2_945 : Bool := FALSE;   // Betriebsmeldungen / Operating messages / Avisos operativos
      User49_DB2_946 : Bool := TRUE;   // UserDataArea 49, DB2.DBB946; Fehlermeldungen / UserDataArea 49, DB2.DBB946; error messages / UserDataArea 49, DB2.DBB946; avisos de error
      User49_DB2_947 : Bool := TRUE;   // Fehlermeldungen / Error messages / Avisos de error
      User49_DB2_948 : Bool := TRUE;   // Fehlermeldungen / Error messages / Avisos de error
      User49_DB2_949 : Bool := TRUE;   // Fehlermeldungen / Error messages / Avisos de error
      User49_DB2_950 : Bool := FALSE;   // Betriebsmeldungen / Operating messages / Avisos operativos
      User49_DB2_951 : Bool := FALSE;   // Betriebsmeldungen / Operating messages / Avisos operativos
      User49_DB2_952 : Bool := FALSE;   // Betriebsmeldungen / Operating messages / Avisos operativos
      User49_DB2_953 : Bool := FALSE;   // Betriebsmeldungen / Operating messages / Avisos operativos
      User50_DB2_954 : Bool := TRUE;   // UserDataArea 50, DB2.DBB954; Fehlermeldungen / UserDataArea 50, DB2.DBB954; error messages / UserDataArea 50, DB2.DBB954; avisos de error
      User50_DB2_955 : Bool := TRUE;   // Fehlermeldungen / Error messages / Avisos de error
      User50_DB2_956 : Bool := TRUE;   // Fehlermeldungen / Error messages / Avisos de error
      User50_DB2_957 : Bool := TRUE;   // Fehlermeldungen / Error messages / Avisos de error
      User50_DB2_958 : Bool := FALSE;   // Betriebsmeldungen / Operating messages / Avisos operativos
      User50_DB2_959 : Bool := FALSE;   // Betriebsmeldungen / Operating messages / Avisos operativos
      User50_DB2_960 : Bool := FALSE;   // Betriebsmeldungen / Operating messages / Avisos operativos
      User50_DB2_961 : Bool := FALSE;   // Betriebsmeldungen / Operating messages / Avisos operativos
      User51_DB2_962 : Bool := TRUE;   // UserDataArea 51, DB2.DBB962; Fehlermeldungen / UserDataArea 51, DB2.DBB962; error messages / UserDataArea 51, DB2.DBB962; avisos de error
      User51_DB2_963 : Bool := TRUE;   // Fehlermeldungen / Error messages / Avisos de error
      User51_DB2_964 : Bool := TRUE;   // Fehlermeldungen / Error messages / Avisos de error
      User51_DB2_965 : Bool := TRUE;   // Fehlermeldungen / Error messages / Avisos de error
      User51_DB2_966 : Bool := FALSE;   // Betriebsmeldungen / Operating messages / Avisos operativos
      User51_DB2_967 : Bool := FALSE;   // Betriebsmeldungen / Operating messages / Avisos operativos
      User51_DB2_968 : Bool := FALSE;   // Betriebsmeldungen / Operating messages / Avisos operativos
      User51_DB2_969 : Bool := FALSE;   // Betriebsmeldungen / Operating messages / Avisos operativos
      User52_DB2_970 : Bool := TRUE;   // UserDataArea 52, DB2.DBB970; Fehlermeldungen / UserDataArea 52, DB2.DBB970; error messages / UserDataArea 52, DB2.DBB970; avisos de error
      User52_DB2_971 : Bool := TRUE;   // Fehlermeldungen / Error messages / Avisos de error
      User52_DB2_972 : Bool := TRUE;   // Fehlermeldungen / Error messages / Avisos de error
      User52_DB2_973 : Bool := TRUE;   // Fehlermeldungen / Error messages / Avisos de error
      User52_DB2_974 : Bool := FALSE;   // Betriebsmeldungen / Operating messages / Avisos operativos
      User52_DB2_975 : Bool := FALSE;   // Betriebsmeldungen / Operating messages / Avisos operativos
      User52_DB2_976 : Bool := FALSE;   // Betriebsmeldungen / Operating messages / Avisos operativos
      User52_DB2_977 : Bool := FALSE;   // Betriebsmeldungen / Operating messages / Avisos operativos
      User53_DB2_978 : Bool := TRUE;   // UserDataArea 53, DB2.DBB978; Fehlermeldungen / UserDataArea 53, DB2.DBB978; error messages / UserDataArea 53, DB2.DBB978; avisos de error
      User53_DB2_979 : Bool := TRUE;   // Fehlermeldungen / Error messages / Avisos de error
      User53_DB2_980 : Bool := TRUE;   // Fehlermeldungen / Error messages / Avisos de error
      User53_DB2_981 : Bool := TRUE;   // Fehlermeldungen / Error messages / Avisos de error
      User53_DB2_982 : Bool := FALSE;   // Betriebsmeldungen / Operating messages / Avisos operativos
      User53_DB2_983 : Bool := FALSE;   // Betriebsmeldungen / Operating messages / Avisos operativos
      User53_DB2_984 : Bool := FALSE;   // Betriebsmeldungen / Operating messages / Avisos operativos
      User53_DB2_985 : Bool := FALSE;   // Betriebsmeldungen / Operating messages / Avisos operativos
      User54_DB2_986 : Bool := TRUE;   // UserDataArea 54, DB2.DBB986; Fehlermeldungen / UserDataArea 54, DB2.DBB986; error messages / UserDataArea 54, DB2.DBB986; avisos de error
      User54_DB2_987 : Bool := TRUE;   // Fehlermeldungen / Error messages / Avisos de error
      User54_DB2_988 : Bool := TRUE;   // Fehlermeldungen / Error messages / Avisos de error
      User54_DB2_989 : Bool := TRUE;   // Fehlermeldungen / Error messages / Avisos de error
      User54_DB2_990 : Bool := FALSE;   // Betriebsmeldungen / Operating messages / Avisos operativos
      User54_DB2_991 : Bool := FALSE;   // Betriebsmeldungen / Operating messages / Avisos operativos
      User54_DB2_992 : Bool := FALSE;   // Betriebsmeldungen / Operating messages / Avisos operativos
      User54_DB2_993 : Bool := FALSE;   // Betriebsmeldungen / Operating messages / Avisos operativos
      User55_DB2_994 : Bool := TRUE;   // UserDataArea 55, DB2.DBB994; Fehlermeldungen / UserDataArea 55, DB2.DBB994; error messages / UserDataArea 55, DB2.DBB994; avisos de error
      User55_DB2_995 : Bool := TRUE;   // Fehlermeldungen / Error messages / Avisos de error
      User55_DB2_996 : Bool := TRUE;   // Fehlermeldungen / Error messages / Avisos de error
      User55_DB2_997 : Bool := TRUE;   // Fehlermeldungen / Error messages / Avisos de error
      User55_DB2_998 : Bool := FALSE;   // Betriebsmeldungen / Operating messages / Avisos operativos
      User55_DB2_999 : Bool := FALSE;   // Betriebsmeldungen / Operating messages / Avisos operativos
      User55_DB2_1000 : Bool := FALSE;   // Betriebsmeldungen / Operating messages / Avisos operativos
      User55_DB2_1001 : Bool := FALSE;   // Betriebsmeldungen / Operating messages / Avisos operativos
      User56_DB2_1002 : Bool := TRUE;   // UserDataArea 56, DB2.DBB1002; Fehlermeldungen / UserDataArea 56, DB2.DBB1002; error messages / UserDataArea 56, DB2.DBB1002; avisos de error
      User56_DB2_1003 : Bool := TRUE;   // Fehlermeldungen / Error messages / Avisos de error
      User56_DB2_1004 : Bool := TRUE;   // Fehlermeldungen / Error messages / Avisos de error
      User56_DB2_1005 : Bool := TRUE;   // Fehlermeldungen / Error messages / Avisos de error
      User56_DB2_1006 : Bool := FALSE;   // Betriebsmeldungen / Operating messages / Avisos operativos
      User56_DB2_1007 : Bool := FALSE;   // Betriebsmeldungen / Operating messages / Avisos operativos
      User56_DB2_1008 : Bool := FALSE;   // Betriebsmeldungen / Operating messages / Avisos operativos
      User56_DB2_1009 : Bool := FALSE;   // Betriebsmeldungen / Operating messages / Avisos operativos
      User57_DB2_1010 : Bool := TRUE;   // UserDataArea 57, DB2.DBB1010; Fehlermeldungen / UserDataArea 57, DB2.DBB1010; error messages / UserDataArea 57, DB2.DBB1010; avisos de error
      User57_DB2_1011 : Bool := TRUE;   // Fehlermeldungen / Error messages / Avisos de error
      User57_DB2_1012 : Bool := TRUE;   // Fehlermeldungen / Error messages / Avisos de error
      User57_DB2_1013 : Bool := TRUE;   // Fehlermeldungen / Error messages / Avisos de error
      User57_DB2_1014 : Bool := FALSE;   // Betriebsmeldungen / Operating messages / Avisos operativos
      User57_DB2_1015 : Bool := FALSE;   // Betriebsmeldungen / Operating messages / Avisos operativos
      User57_DB2_1016 : Bool := FALSE;   // Betriebsmeldungen / Operating messages / Avisos operativos
      User57_DB2_1017 : Bool := FALSE;   // Betriebsmeldungen / Operating messages / Avisos operativos
      User58_DB2_1018 : Bool := TRUE;   // UserDataArea 58, DB2.DBB1018; Fehlermeldungen / UserDataArea 58, DB2.DBB1018; error messages / UserDataArea 58, DB2.DBB1018; avisos de error
      User58_DB2_1019 : Bool := TRUE;   // Fehlermeldungen / Error messages / Avisos de error
      User58_DB2_1020 : Bool := TRUE;   // Fehlermeldungen / Error messages / Avisos de error
      User58_DB2_1021 : Bool := TRUE;   // Fehlermeldungen / Error messages / Avisos de error
      User58_DB2_1022 : Bool := FALSE;   // Betriebsmeldungen / Operating messages / Avisos operativos
      User58_DB2_1023 : Bool := FALSE;   // Betriebsmeldungen / Operating messages / Avisos operativos
      User58_DB2_1024 : Bool := FALSE;   // Betriebsmeldungen / Operating messages / Avisos operativos
      User58_DB2_1025 : Bool := FALSE;   // Betriebsmeldungen / Operating messages / Avisos operativos
      User59_DB2_1026 : Bool := TRUE;   // UserDataArea 59, DB2.DBB1026; Fehlermeldungen / UserDataArea 59, DB2.DBB1026; error messages / UserDataArea 59, DB2.DBB1026; avisos de error
      User59_DB2_1027 : Bool := TRUE;   // Fehlermeldungen / Error messages / Avisos de error
      User59_DB2_1028 : Bool := TRUE;   // Fehlermeldungen / Error messages / Avisos de error
      User59_DB2_1029 : Bool := TRUE;   // Fehlermeldungen / Error messages / Avisos de error
      User59_DB2_1030 : Bool := FALSE;   // Betriebsmeldungen / Operating messages / Avisos operativos
      User59_DB2_1031 : Bool := FALSE;   // Betriebsmeldungen / Operating messages / Avisos operativos
      User59_DB2_1032 : Bool := FALSE;   // Betriebsmeldungen / Operating messages / Avisos operativos
      User59_DB2_1033 : Bool := FALSE;   // Betriebsmeldungen / Operating messages / Avisos operativos
      User60_DB2_1034 : Bool := TRUE;   // UserDataArea 60, DB2.DBB1034; Fehlermeldungen / UserDataArea 60, DB2.DBB1034; error messages / UserDataArea 60, DB2.DBB1034; avisos de error
      User60_DB2_1035 : Bool := TRUE;   // Fehlermeldungen / Error messages / Avisos de error
      User60_DB2_1036 : Bool := TRUE;   // Fehlermeldungen / Error messages / Avisos de error
      User60_DB2_1037 : Bool := TRUE;   // Fehlermeldungen / Error messages / Avisos de error
      User60_DB2_1038 : Bool := FALSE;   // Betriebsmeldungen / Operating messages / Avisos operativos
      User60_DB2_1039 : Bool := FALSE;   // Betriebsmeldungen / Operating messages / Avisos operativos
      User60_DB2_1040 : Bool := FALSE;   // Betriebsmeldungen / Operating messages / Avisos operativos
      User60_DB2_1041 : Bool := FALSE;   // Betriebsmeldungen / Operating messages / Avisos operativos
      User61_DB2_1042 : Bool := TRUE;   // UserDataArea 61, DB2.DBB1042; Fehlermeldungen / UserDataArea 61, DB2.DBB1042; error messages / UserDataArea 61, DB2.DBB1042; avisos de error
      User61_DB2_1043 : Bool := TRUE;   // Fehlermeldungen / Error messages / Avisos de error
      User61_DB2_1044 : Bool := TRUE;   // Fehlermeldungen / Error messages / Avisos de error
      User61_DB2_1045 : Bool := TRUE;   // Fehlermeldungen / Error messages / Avisos de error
      User61_DB2_1046 : Bool := FALSE;   // Betriebsmeldungen / Operating messages / Avisos operativos
      User61_DB2_1047 : Bool := FALSE;   // Betriebsmeldungen / Operating messages / Avisos operativos
      User61_DB2_1048 : Bool := FALSE;   // Betriebsmeldungen / Operating messages / Avisos operativos
      User61_DB2_1049 : Bool := FALSE;   // Betriebsmeldungen / Operating messages / Avisos operativos
      User62_DB2_1050 : Bool := TRUE;   // UserDataArea 62, DB2.DBB1050; Fehlermeldungen / UserDataArea 62, DB2.DBB1050; error messages / UserDataArea 62, DB2.DBB1050; avisos de error
      User62_DB2_1051 : Bool := TRUE;   // Fehlermeldungen / Error messages / Avisos de error
      User62_DB2_1052 : Bool := TRUE;   // Fehlermeldungen / Error messages / Avisos de error
      User62_DB2_1053 : Bool := TRUE;   // Fehlermeldungen / Error messages / Avisos de error
      User62_DB2_1054 : Bool := FALSE;   // Betriebsmeldungen / Operating messages / Avisos operativos
      User62_DB2_1055 : Bool := FALSE;   // Betriebsmeldungen / Operating messages / Avisos operativos
      User62_DB2_1056 : Bool := FALSE;   // Betriebsmeldungen / Operating messages / Avisos operativos
      User62_DB2_1057 : Bool := FALSE;   // Betriebsmeldungen / Operating messages / Avisos operativos
      User63_DB2_1058 : Bool := TRUE;   // UserDataArea 63, DB2.DBB1058; Fehlermeldungen / UserDataArea 63, DB2.DBB1058; error messages / UserDataArea 63, DB2.DBB1058; avisos de error
      User63_DB2_1059 : Bool := TRUE;   // Fehlermeldungen / Error messages / Avisos de error
      User63_DB2_1060 : Bool := TRUE;   // Fehlermeldungen / Error messages / Avisos de error
      User63_DB2_1061 : Bool := TRUE;   // Fehlermeldungen / Error messages / Avisos de error
      User63_DB2_1062 : Bool := FALSE;   // Betriebsmeldungen / Operating messages / Avisos operativos
      User63_DB2_1063 : Bool := FALSE;   // Betriebsmeldungen / Operating messages / Avisos operativos
      User63_DB2_1064 : Bool := FALSE;   // Betriebsmeldungen / Operating messages / Avisos operativos
      User63_DB2_1065 : Bool := FALSE;   // Betriebsmeldungen / Operating messages / Avisos operativos
   END_VAR
BEGIN
END_DATA_BLOCK
